// Mitsubishi GX Works2 project: 260625타이머   PLC: Q02/Q02H

PROGRAM MAIN
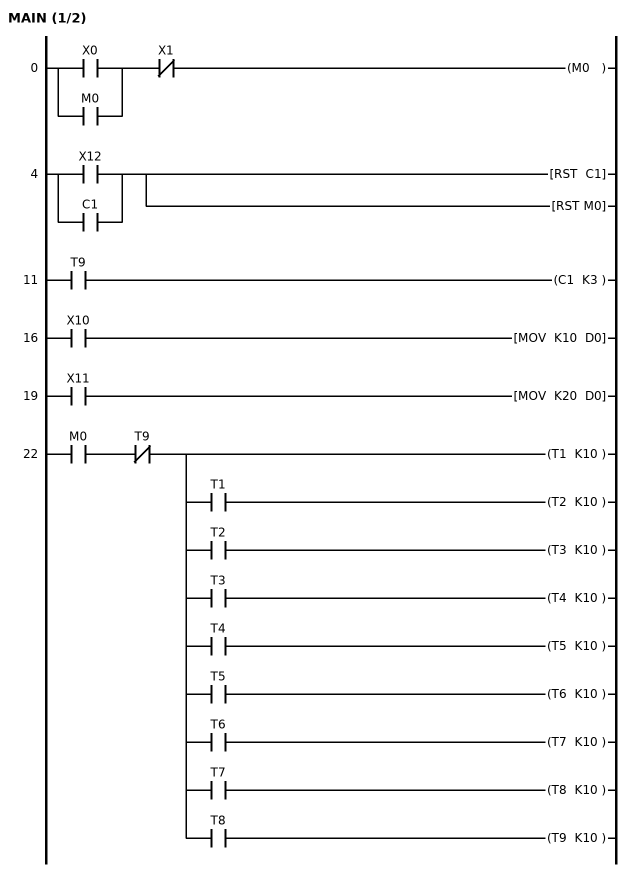
0     LD      X0
      OR      M0
      ANI     X1
      OUT     M0
4     LD      X12
      OR      C1
      RST     C1
      RST     M0
11    LD      T9
      OUT     C1 K3
16    LD      X10
      MOV     K10 D0
19    LD      X11
      MOV     K20 D0
22    LD      M0
      ANI     T9
      OUT     T1 K10
      MPS
      AND     T1
      OUT     T2 K10
      MRD
      AND     T2
      OUT     T3 K10
      MRD
      AND     T3
      OUT     T4 K10
      MRD
      AND     T4
      OUT     T5 K10
      MRD
      AND     T5
      OUT     T6 K10
      MRD
      AND     T6
      OUT     T7 K10
      MRD
      AND     T7
      OUT     T8 K10
      MPP
      AND     T8
      OUT     T9 K10
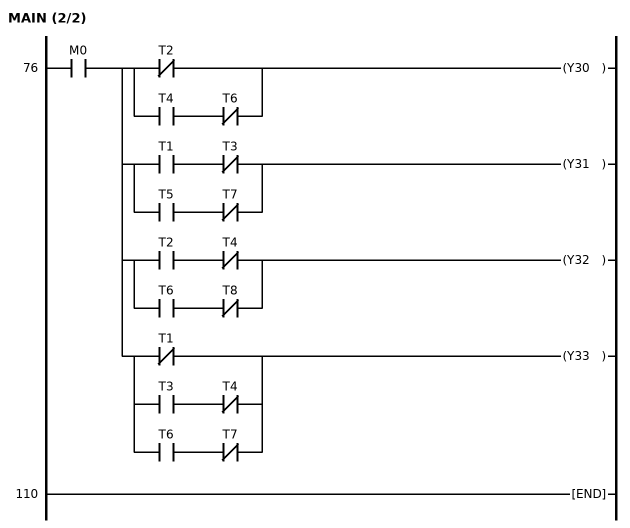
76    LD      M0
      MPS
      LDI     T2
      LD      T4
      ANI     T6
      ORB
      ANB
      OUT     Y30
      MRD
      LD      T1
      ANI     T3
      LD      T5
      ANI     T7
      ORB
      ANB
      OUT     Y31
      MRD
      LD      T2
      ANI     T4
      LD      T6
      ANI     T8
      ORB
      ANB
      OUT     Y32
      MPP
      LDI     T1
      LD      T3
      ANI     T4
      ORB
      LD      T6
      ANI     T7
      ORB
      ANB
      OUT     Y33
110   END
END_PROGRAM
